// TIA Portal V20 export
TYPE "LKinCtrl_typeCOffInCurrentPos"
   STRUCT
      positionAbsolute : "LKinCtrl_typeCartesianPosition";   // Source data - current absolute position
      positionAbsoluteRadComp : "LKinCtrl_typeCartesianPosition";   // Source data - current absolute position radius compensated
   END_STRUCT;
END_TYPE
